// TwinCAT 3 PLC project Library
// Title: lcls-twincat-sample-delivery
// Company: SLAC
// ProjectVersion: 1.0.0
// ProgramVersion: 3.1.4023.0
// libraries:
//   LCLS General, * (SLAC)
//   LCLS Vacuum, * (SLAC - LCLS)
//   PMPS, * (SLAC - LCLS)
//   Tc2_EtherCAT, * (Beckhoff Automation GmbH)
//   Tc2_MC2, * (Beckhoff Automation GmbH)
//   Tc2_ModbusSrv, * (Beckhoff Automation GmbH)
//   Tc2_SerialCom, * (Beckhoff Automation GmbH)
//   Tc2_Standard, * (Beckhoff Automation GmbH)
//   Tc2_SUPS, * (Beckhoff Automation GmbH)
//   Tc2_System, * (Beckhoff Automation GmbH)
//   Tc2_Utilities, * (Beckhoff Automation GmbH)
//   Tc3_Module, * (Beckhoff Automation GmbH)
//   TcUnit, * (www.tcunit.org)
// project tree:
//   DUTs/ALI/ E_AxisMoveMode.TcDUT (not stored), E_CTRL_MODE.TcDUT (not stored), E_PropValveFBState.TcDUT (not stored), HMI_PropValveCtrlState.TcDUT (not stored), ST_ALI.TcDUT (not stored), ST_ManipAxis.TcDUT (not stored), ST_PIDParams.TcDUT (not stored), ST_PressureController.TcDUT (not stored), ST_PropValveMKS253.TcDUT (not stored)
//   DUTs/Bronkhorst/ E_BHElFlowUnit.TcDUT (not stored), ST_BhElFlow.TcDUT (not stored)
//   DUTs/ E_AxisMotionState.TcDUT (not stored), ST_ManifoldValve.TcDUT (not stored), ST_Proportionair.TcDUT (not stored), ST_RegDeadbandControls.TcDUT (not stored), ST_Regulator.TcDUT (not stored), ST_SelectorM3.TcDUT (not stored), ST_Shaker.TcDUT (not stored), ST_ShakerControls.TcDUT (not stored), ST_Strings.TcDUT (not stored)
//   DUTs/General/ E_CTRL_MODE_1.TcDUT
//   DUTs/IO_Structs/ ST_ALIIO.TcDUT (not stored), ST_M3DeviceBaseIO.TcDUT (not stored), ST_SerialComm.TcDUT (not stored)
//   DUTs/Sensirion/ E_SensirionFMMode.TcTLEO (not stored), ST_SensirionFM.TcDUT (not stored), ST_SensirionFMControl.TcDUT (not stored), ST_SensirionFMStatus.TcDUT (not stored)
//   DUTs/TEC/ ST_TECControl.TcDUT (not stored), ST_TECStatus.TcDUT (not stored)
//   DUTs/Vici/ ST_4PViciValveSampleNames.TcDUT, ST_ViciControl.TcDUT (not stored), ST_ViciStatus.TcDUT (not stored)
//   GVLs/ GVL_SAMPLE.TcGVL
//   / PlcTask.TcTTO
//   POUs/ALI/ FB_ALI.TcPOU (not stored), FB_ManipAxis.TcPOU (not stored), FB_PID_EXT.TcPOU (not stored), FB_PropValve.TcPOU (not stored), F_AxisRef_To_MSTA.TcPOU (not stored), MC_SmoothMover.TcPOU (not stored)
//   POUs/Bronkhorst/ FB_BronkhorstMFM.TcPOU (not stored)
//   POUs/DigitalOutput/ FB_SolenoidPair.TcPOU (not stored)
//   POUs/ FB_RCC.TcPOU, EXAMPLE_DEPLOYMENT.TcPOU (not stored), PRG_TEST.TcPOU (not stored)
//   POUs/GasManifold/ FB_GasManifold.TcPOU (not stored), FB_ManiValve.TcPOU (not stored)
//   POUs/Helpers/ FB_EcatDiag.TcPOU (not stored), FB_SelectorSync.TcPOU (not stored), FB_SerialCommWrapper.TcPOU (not stored), FB_ShiftByteArray.TcPOU (not stored)
//   POUs/PCM/ FB_PressureControlModule.TcPOU (not stored)
//   POUs/Regulators/ FB_ProportionairRegulator.TcPOU (not stored), FB_Regulator.TcPOU (not stored), F_rPressure.TcPOU (not stored)
//   POUs/Selectors/ FB_SelectorM3.TcPOU (not stored)
//   POUs/Sensirion/ FB_SensirionDriver.TcPOU, FB_SensirionTransaction.TcPOU (not stored), fSHDLCChecksum.TcPOU (not stored)
//   POUs/TEC/ FB_TECDriver.TcPOU (not stored), FB_TECTransaction.TcPOU (not stored)
//   POUs/Tests/ FB_RCC_TEST.TcPOU
//   POUs/VICI/ FB_4PortViciValve.TcPOU, FB_ViciDriver.TcPOU, FB_ViciTransaction.TcPOU (not stored), FB_ViciValve.TcPOU (not stored)

CONFIGURATION Library
    RESOURCE PLC ON TwinCAT3
        TASK PlcTask(INTERVAL := T#10ms, PRIORITY := 20);
        PROGRAM PRG_TEST WITH PlcTask : PRG_TEST;
    END_RESOURCE
END_CONFIGURATION

// ---- DUTs/General/E_CTRL_MODE_1.TcDUT
{attribute 'qualified_only'}
{attribute 'strict'}
TYPE E_CTRL_MODE_1 :
(
    enum_member := 0
);
END_TYPE

// ---- DUTs/Vici/ST_4PViciValveSampleNames.TcDUT
TYPE ST_4PViciValveSampleNames :
STRUCT
      {attribute 'pytmc' := '
        pv: 01
        io: io
     '}
     s1 : STRING;
     {attribute 'pytmc' := '
        pv: 02
        io: io
     '}
     s2 : STRING;
     {attribute 'pytmc' := '
        pv: 03
        io: io
     '}
     s3 : STRING;
     {attribute 'pytmc' := '
        pv: 04
        io: io
     '}
     s4 : STRING;
END_STRUCT
END_TYPE

// ---- GVLs/GVL_SAMPLE.TcGVL
VAR_GLOBAL
    g_xFirstPass: BOOL := TRUE;
END_VAR

// ---- POUs/FB_RCC.TcPOU
FUNCTION_BLOCK FB_RCC
VAR_IN_OUT
	RCC_VRC_01 : FB_VRC_NC_ClsLS;
	RCC_VRC_02 : FB_VRC;
	RCC_VRC_03 : FB_VRC_NC_ClsLS;
	RCC_VRC_04 : FB_VRC_NC_ClsLS;
	RCC_GCP_01 : FB_901_ECAT;
END_VAR
VAR
	{attribute 'pytmc' :=' pv: ILK_Setpoint '}
    RCC_GCP_01_INTERLOCK_SETPOINT : REAL := 10;
	{attribute 'pytmc' :=' pv: OverrideMode '}
	xSystemOverrideMode_RCC : BOOL := FALSE;
	{attribute 'pytmc' :=' pv: sLogMessage '}
	sLogMessage : T_MaxString := "";
	fbFormat   : FB_FormatString;
	
	tTimer1 : TON;
	current_state : INT := 0;
	start_cycle : BOOL  := FALSE;
	
	RCC_VRC_01_OPEN_OK : BOOL;
    RCC_VRC_02_OPEN_OK : BOOL;
    RCC_VRC_03_OPEN_OK : BOOL;
    RCC_VRC_04_OPEN_OK : BOOL;
END_VAR


(* Valve can open only when CRIX-RCC-VRC-02 and 03 are closed*)
RCC_VRC_01_OPEN_OK := ( RCC_VRC_02.iq_stValve.i_xClsLS AND NOT RCC_VRC_02.iq_stValve.q_xOPN_DO ) AND
                                    ( RCC_VRC_03.iq_stValve.i_xClsLS AND NOT RCC_VRC_03.iq_stValve.q_xOPN_DO ) ;

RCC_VRC_01(i_xExtILK_OK := RCC_VRC_01_OPEN_OK,
                i_xOverrideMode := xSystemOverrideMode_RCC,
                 iq_stValve=> );

(* Valve can open only when CRIX-RCC-VRC-01 and 04 are closed*)
RCC_VRC_02_OPEN_OK := ( RCC_VRC_01.iq_stValve.i_xClsLS AND NOT RCC_VRC_01.iq_stValve.q_xOPN_DO ) AND
                                    ( RCC_VRC_04.iq_stValve.i_xClsLS AND NOT RCC_VRC_04.iq_stValve.q_xOPN_DO );

RCC_VRC_02(i_xExtILK_OK := RCC_VRC_02_OPEN_OK,
                i_xOverrideMode := xSystemOverrideMode_RCC,
                 iq_stValve=> );

(* Valve can open only when CRIX-RCC-GCP-01 reading < setpoint Torr and CRIX-RCC-VRC-01 and 04 are closed*)
RCC_VRC_03_OPEN_OK := (RCC_GCP_01.PG.rPRESS < RCC_GCP_01_INTERLOCK_SETPOINT and RCC_GCP_01.PG.xPRESS_OK ) AND
                                 ( RCC_VRC_01.iq_stValve.i_xClsLS AND NOT RCC_VRC_01.iq_stValve.q_xOPN_DO ) AND
                                              ( RCC_VRC_04.iq_stValve.i_xClsLS AND NOT RCC_VRC_04.iq_stValve.q_xOPN_DO );

RCC_VRC_03(i_xExtILK_OK := RCC_VRC_03_OPEN_OK,
                i_xOverrideMode := xSystemOverrideMode_RCC,
                 iq_stValve=> );

(* Valve can open only when CRIX-RCC-VRC-02 and 03 are closed*)
RCC_VRC_04_OPEN_OK := ( RCC_VRC_02.iq_stValve.i_xClsLS AND NOT RCC_VRC_02.iq_stValve.q_xOPN_DO ) AND
                                      ( RCC_VRC_03.iq_stValve.i_xClsLS AND NOT RCC_VRC_03.iq_stValve.q_xOPN_DO ) ;

RCC_VRC_04(i_xExtILK_OK := RCC_VRC_04_OPEN_OK,
                i_xOverrideMode := xSystemOverrideMode_RCC,
                 iq_stValve=> );

METHOD PUBLIC cycle : BOOL
VAR_INPUT
	t1 : TIME := T#20s;
	t2 : TIME := T#10s;
	t3 : TIME := T#5s;
	t4 : TIME := T#10s;
	run_clean : BOOL := TRUE;
END_VAR
CASE current_state OF
	-1:
		IF start_cycle THEN 
			current_state := 0; 
			start_cycle := FALSE;
		END_IF
		
	0:
		RCC_VRC_01.iq_stValve.q_xOPN_DO := FALSE;
		RCC_VRC_02.iq_stValve.q_xOPN_DO := FALSE;
		RCC_VRC_03.iq_stValve.q_xOPN_DO := FALSE;
		RCC_VRC_04.iq_stValve.q_xOPN_DO := FALSE;
		current_state:=1;
		
	1: // OPEN
		tTimer1(IN:=TRUE, PT:=t1);
		RCC_VRC_02.iq_stValve.q_xOPN_DO := TRUE;
	
		IF tTimer1.Q THEN 
			current_state := 2;
			tTimer1(IN:=FALSE); // RESTART TIMER
		END_IF
		
	2:	// DRAIN_1
		IF RCC_VRC_03_OPEN_OK THEN 
			IF run_clean THEN RCC_VRC_02.iq_stValve.q_xOPN_DO := FALSE; END_IF
			RCC_VRC_03.iq_stValve.q_xOPN_DO := TRUE;
			current_state := 3; 
		END_IF
		
	3:	// DRAIN_2
		tTimer1(IN:=TRUE, PT:=t2);
		
		IF tTimer1.Q THEN 
			current_state := 4;
			IF NOT RCC_VRC_03_OPEN_OK THEN current_state := 1; END_IF
 			RCC_VRC_03.iq_stValve.q_xOPN_DO := FALSE;
			IF NOT run_clean THEN RCC_VRC_02.iq_stValve.q_xOPN_DO := FALSE; END_IF
			tTimer1(IN:=FALSE); // RESTART TIMER
		END_IF
		
	4: // OPEN VRC_01 for T3
		tTimer1(IN:=TRUE, PT:=t3);
		RCC_VRC_01.iq_stValve.q_xOPN_DO := TRUE;
		IF tTimer1.Q THEN 
			current_state := 5;
			tTimer1(IN:=FALSE); // RESTART TIMER
		END_IF
		
	5: // OPEN VRC_04 for T4
		tTimer1(IN:=TRUE, PT:=t4);
		RCC_VRC_04.iq_stValve.q_xOPN_DO := TRUE;
		IF tTimer1.Q THEN 
			current_state := -1;
			RCC_VRC_01.iq_stValve.q_xOPN_DO := FALSE;
			RCC_VRC_04.iq_stValve.q_xOPN_DO := FALSE;
			tTimer1(IN:=FALSE); // RESTART TIMER
		END_IF	
	
	
END_CASE
END_METHOD

END_FUNCTION_BLOCK

// ---- POUs/Sensirion/FB_SensirionDriver.TcPOU
FUNCTION_BLOCK FB_SensirionDriver

VAR_INPUT
    i_xExecute				: BOOL := FALSE;		(* rising edge execute *)
    i_tTimeOut				: TIME := T#10S;  		(* Maximum wait time for reply *)
    i_stControl				: ST_SensirionFMControl;
END_VAR
VAR_OUTPUT
    q_xDone					: BOOL;
    q_xError				: BOOL;
    q_xWarning				: BOOL;					(* set in the event of an unexpected reply *)
    q_xTimeout				: BOOL;
    q_asResult				: ARRAY[1..60] OF STRING(255);
    q_stStatus				: ST_SensirionFMStatus;
    q_xInitComplete			: BOOL;
END_VAR
VAR_IN_OUT
    iq_stSerialRXBuffer 	: ComBuffer;
    iq_stSerialTXBuffer 	: ComBuffer;
END_VAR
VAR
    //Usual stuff
    rtExecute				: R_TRIG;
    rtReInit				:	R_TRIG;
    iStep					: INT;
    iResultIndex			:	INT := 1;
    aiSteps	:	ARRAY[1..256] OF INT;
    iStepIndex	:	INT;
    fbSensirionTransaction		: FB_SensirionTransaction;

    //Device Specific Working Variables
    tonDelay : TON;
    bLen	:	BYTE;
    abTxData	:	ARRAY[1..256] OF BYTE;
    xInitComplete	:	BOOL;
    abRxData	:	ARRAY[1..256] OF BYTE;

    iScale	:	INT;
    iUnit	:	INT;
    xType	:	BOOL;
    xMode	:	BYTE;
    xLinear	:	BOOL;
    uiOffset	:	UINT;
    iIdleAttempt : INT;

    //Command delays
    tonCommandDelay : TON;
xcatch : BOOL;
END_VAR

(* This function block performs serial communication with a Sensirion meter *)


(* rising edge trigger *)
rtExecute(CLK:= i_xExecute);
rtReInit(CLK:= i_stControl.xReset);
IF rtReInit.Q THEN xInitComplete := FALSE; END_IF
IF rtExecute.Q  THEN
    q_xDone	:= FALSE;
    q_xError := FALSE;
    q_xWarning := FALSE;
    q_xTimeout := FALSE;
    q_asResult[iResultIndex]:= '';
    fbSensirionTransaction( i_xExecute:= FALSE, iq_stSerialRXBuffer:= iq_stSerialRXBuffer, iq_stSerialTXBuffer:= iq_stSerialTXBuffer );  (* reset *)
    IF xInitComplete THEN
        iStep := 30;
        (* Branch to reset device if reset bit is set here *)
        IF rtReInit.Q  OR (i_stControl.xCalMode <> q_stStatus.xFMMode) THEN
            iStep := 400;
            xInitComplete := FALSE;
            q_stStatus.xFlowValid := FALSE;
            q_asResult[iResultIndex] := 'Reinitializing';
            iResultIndex := iResultIndex +1;
        END_IF
    ELSIF i_stControl.xReset THEN
        iStep := 400;
        q_stStatus.xFlowValid := FALSE;
        q_asResult[iResultIndex] := 'Reinitializing';
        iResultIndex := iResultIndex +1;
    ELSE
        iStep := 9;
    END_IF
END_IF

CASE iStep OF
    0: (* idle *)
        ;

    9: //Get cal mode
    fbSensirionTransaction(
        i_xExecute:= TRUE,
        i_bAdr:= i_stControl.bAdr,
        i_bLen:= 0,
        i_bCmd:= 16#43,
        i_abTxData := abTxData,
        i_tTimeOut:= i_tTimeOut,
        iq_stSerialRXBuffer:= iq_stSerialRXBuffer,
        iq_stSerialTXBuffer:= iq_stSerialTXBuffer
        );
    IF fbSensirionTransaction.q_xError THEN
        q_asResult[iResultIndex] := CONCAT('in Step 9 serial transaction failed with message: ', fbSensirionTransaction.q_sResult);
        iResultIndex := iResultIndex +1;
        iStep := 9000;
    ELSIF fbSensirionTransaction.q_xDone THEN
        //abRxdata := fbSensirionTransaction.q_baRxData;
        IF UDINT_TO_BOOL(MEMCPY(destAddr:=ADR(xMode), srcAddr:=ADR(fbSensirionTransaction.q_baRxData), n:=1)) THEN
            q_stStatus.xFMMode := BYTE_TO_BOOL(xMode);
            fbSensirionTransaction( i_xExecute:= FALSE, iq_stSerialRXBuffer:= iq_stSerialRXBuffer, iq_stSerialTXBuffer:= iq_stSerialTXBuffer );  (* reset *)
            q_asResult[iResultIndex] := CONCAT('Step 9 complete. Cal mode is set to: ', BYTE_TO_STRING(xMode));
            iResultIndex := iResultIndex +1;
        ELSE
            iStep := 9000;
            q_asResult[iResultIndex] := 'Memcpy in step 9 failed';
            iResultIndex := iResultIndex +1;
        END_IF
        iStep := 10;
    END_IF

    10: // Set calibration
    //calibration of 0 for precision mode, 250 nL/min - 5000 nL/min
    // calibration of 1 for extended mode, 2000 nL/min - 20000 nL/min
    IF q_stStatus.xFMMode <> i_stControl.xCalMode THEN
        IF i_stControl.xCalMode THEN abTxData[1]:=1; ELSE abTxData[1]:=0; END_IF
        fbSensirionTransaction(
            i_xExecute:= TRUE,
            i_bAdr:= i_stControl.bAdr,
            i_bLen:= 1,
            i_bCmd:= 16#43,
            i_abTxData := abTxData,
            i_tTimeOut:= i_tTimeOut,
            iq_stSerialRXBuffer:= iq_stSerialRXBuffer,
            iq_stSerialTXBuffer:= iq_stSerialTXBuffer
            );
        IF fbSensirionTransaction.q_xError THEN
            q_asResult[iResultIndex] := CONCAT('in Step 10 serial transaction failed with message: ', fbSensirionTransaction.q_sResult);
            iResultIndex := iResultIndex +1;
            iStep := 9000;
        ELSIF fbSensirionTransaction.q_xDone THEN
            tonCommandDelay(IN:=fbSensirionTransaction.q_xDone, PT:=T#1S);
            IF tonCommandDelay.Q THEN
                (* No response, completed transaction confirmed by a response*)
                q_asResult[iResultIndex] := 'Step 10 complete';
                iResultIndex := iResultIndex +1;
                iStep := 11;
                fbSensirionTransaction( i_xExecute:= FALSE, iq_stSerialRXBuffer:= iq_stSerialRXBuffer, iq_stSerialTXBuffer:= iq_stSerialTXBuffer );  (* reset *)
            END_IF
        END_IF
    ELSE
        q_asResult[iResultIndex] := 'Calmode already set';
        iResultIndex := iResultIndex +1;
        iStep := 11;
    END_IF

    11: //Get cal mode
    fbSensirionTransaction(
        i_xExecute:= TRUE,
        i_bAdr:= i_stControl.bAdr,
        i_bLen:= 0,
        i_bCmd:= 16#43,
        i_abTxData := abTxData,
        i_tTimeOut:= i_tTimeOut,
        iq_stSerialRXBuffer:= iq_stSerialRXBuffer,
        iq_stSerialTXBuffer:= iq_stSerialTXBuffer
        );
    IF fbSensirionTransaction.q_xError THEN
        q_asResult[iResultIndex] := CONCAT('in Step 11 serial transaction failed with message: ', fbSensirionTransaction.q_sResult);
        iResultIndex := iResultIndex +1;
        iStep := 9000;
    ELSIF fbSensirionTransaction.q_bState <> 0 THEN
        q_asResult[iResultIndex] := CONCAT('in Step 11 serial transaction failed with error state: ', BYTE_TO_STRING(fbSensirionTransaction.q_bState));
        iResultIndex := iResultIndex +1;
        fbSensirionTransaction( i_xExecute:= FALSE, iq_stSerialRXBuffer:= iq_stSerialRXBuffer, iq_stSerialTXBuffer:= iq_stSerialTXBuffer );  (* reset *)
        iStep := 9000;
    ELSIF fbSensirionTransaction.q_xDone THEN
        tonCommandDelay(IN:=fbSensirionTransaction.q_xDone, PT:=T#100MS);
        IF tonCommandDelay.Q THEN
            IF UDINT_TO_BOOL(MEMCPY(destAddr:=ADR(xMode), srcAddr:=ADR(fbSensirionTransaction.q_baRxData), n:=1)) THEN
                q_stStatus.xFMMode := BYTE_TO_BOOL(xMode);
                fbSensirionTransaction( i_xExecute:= FALSE, iq_stSerialRXBuffer:= iq_stSerialRXBuffer, iq_stSerialTXBuffer:= iq_stSerialTXBuffer );  (* reset *)
                q_asResult[iResultIndex] := 'Step 11 complete';
                iResultIndex := iResultIndex +1;
                iStep := 12;
            ELSE
                iStep := 9000;
                q_asResult[iResultIndex] := 'Memcpy in step 9 failed';
                iResultIndex := iResultIndex +1;
            END_IF
        END_IF
    END_IF

    12: //Get scale factor
    fbSensirionTransaction(
        i_xExecute:= TRUE,
        i_bAdr:= i_stControl.bAdr,
        i_bLen:= 0,
        i_bCmd:= 16#53,
        i_abTxData := abTxData,
        i_tTimeOut:= i_tTimeOut,
        iq_stSerialRXBuffer:= iq_stSerialRXBuffer,
        iq_stSerialTXBuffer:= iq_stSerialTXBuffer
        );
    IF fbSensirionTransaction.q_xError THEN
        q_asResult[iResultIndex] := CONCAT('in Step 12 serial transaction failed with message: ', fbSensirionTransaction.q_sResult);
        iResultIndex := iResultIndex +1;
        iStep := 9000;
    ELSIF fbSensirionTransaction.q_bState <> 0 THEN
        q_asResult[iResultIndex] := CONCAT('in Step 12 serial transaction failed with error state: ', BYTE_TO_STRING(fbSensirionTransaction.q_bState));
        iResultIndex := iResultIndex +1;
        fbSensirionTransaction( i_xExecute:= FALSE, iq_stSerialRXBuffer:= iq_stSerialRXBuffer, iq_stSerialTXBuffer:= iq_stSerialTXBuffer );  (* reset *)
        iStep := 9000;
    ELSIF fbSensirionTransaction.q_xDone THEN
        tonCommandDelay(IN:=fbSensirionTransaction.q_xDone, PT:=T#100MS);
        IF tonCommandDelay.Q THEN
            IF UDINT_TO_BOOL(MEMCPY(destAddr:=ADR(iScale), srcAddr:=ADR(fbSensirionTransaction.q_baRxData), n:=2)) THEN //always 2 for the 16 bit wide integer
                iScale := WORD_TO_INT(HOST_TO_BE16(INT_TO_WORD(iScale)));
                fbSensirionTransaction( i_xExecute:= FALSE, iq_stSerialRXBuffer:= iq_stSerialRXBuffer, iq_stSerialTXBuffer:= iq_stSerialTXBuffer );  (* reset *)
                q_asResult[iResultIndex] := 'Step 12 complete';
                iResultIndex := iResultIndex +1;
                iStep := 13;
            ELSE
                iStep := 9000;
                q_asResult[iResultIndex] := 'Memcpy in step 12 failed';
                iResultIndex := iResultIndex +1;
            END_IF
        END_IF
    END_IF

    13: //Get flow unit
    fbSensirionTransaction(
        i_xExecute:= TRUE,
        i_bAdr:= i_stControl.bAdr,
        i_bLen:= 0,
        i_bCmd:= 16#52,
        i_abTxData := abTxData,
        i_tTimeOut:= i_tTimeOut,
        iq_stSerialRXBuffer:= iq_stSerialRXBuffer,
        iq_stSerialTXBuffer:= iq_stSerialTXBuffer
        );
    IF fbSensirionTransaction.q_xError THEN
        q_asResult[iResultIndex] := CONCAT('in Step 13 serial transaction failed with message: ', fbSensirionTransaction.q_sResult);
        iResultIndex := iResultIndex +1;
        iStep := 9000;
    ELSIF fbSensirionTransaction.q_bState <> 0 THEN
        q_asResult[iResultIndex] := CONCAT('in Step 13 serial transaction failed with error state: ', BYTE_TO_STRING(fbSensirionTransaction.q_bState));
        iResultIndex := iResultIndex +1;
        fbSensirionTransaction( i_xExecute:= FALSE, iq_stSerialRXBuffer:= iq_stSerialRXBuffer, iq_stSerialTXBuffer:= iq_stSerialTXBuffer );  (* reset *)
        iStep := 9000;
    ELSIF fbSensirionTransaction.q_xDone THEN
        tonCommandDelay(IN:=fbSensirionTransaction.q_xDone, PT:=T#100MS);
        IF tonCommandDelay.Q THEN
            IF UDINT_TO_BOOL(MEMCPY(destAddr:=ADR(iUnit), srcAddr:=ADR(fbSensirionTransaction.q_baRxData), n:=2)) THEN //always 2 for the 16 bit wide integer
                iUnit := WORD_TO_INT(HOST_TO_BE16(INT_TO_WORD(iUnit)));
                fbSensirionTransaction( i_xExecute:= FALSE, iq_stSerialRXBuffer:= iq_stSerialRXBuffer, iq_stSerialTXBuffer:= iq_stSerialTXBuffer );  (* reset *)
                q_asResult[iResultIndex] := 'Step 13 complete';
                iResultIndex := iResultIndex +1;
                iStep := 14;
            ELSE
                iStep := 9000;
                q_asResult[iResultIndex] := 'Memcpy in step 13 failed';
                iResultIndex := iResultIndex +1;
            END_IF
        END_IF
    END_IF

    14: //Get measurement type
    fbSensirionTransaction(
        i_xExecute:= TRUE,
        i_bAdr:= i_stControl.bAdr,
        i_bLen:= 0,
        i_bCmd:= 16#55,
        i_abTxData := abTxData,
        i_tTimeOut:= i_tTimeOut,
        iq_stSerialRXBuffer:= iq_stSerialRXBuffer,
        iq_stSerialTXBuffer:= iq_stSerialTXBuffer
        );
    IF fbSensirionTransaction.q_xError THEN
        q_asResult[iResultIndex] := CONCAT('in Step 14 serial transaction failed with message: ', fbSensirionTransaction.q_sResult);
        iResultIndex := iResultIndex +1;
        iStep := 9000;
    ELSIF fbSensirionTransaction.q_bState <> 0 THEN
        q_asResult[iResultIndex] := CONCAT('in Step 14 serial transaction failed with error state: ', BYTE_TO_STRING(fbSensirionTransaction.q_bState));
        iResultIndex := iResultIndex +1;
        fbSensirionTransaction( i_xExecute:= FALSE, iq_stSerialRXBuffer:= iq_stSerialRXBuffer, iq_stSerialTXBuffer:= iq_stSerialTXBuffer );  (* reset *)
        iStep := 9000;
    ELSIF fbSensirionTransaction.q_xDone THEN
        tonCommandDelay(IN:=fbSensirionTransaction.q_xDone, PT:=T#100MS);
        IF tonCommandDelay.Q THEN
            xType := BYTE_TO_BOOL(fbSensirionTransaction.q_baRxData[1]);
            q_asResult[iResultIndex] := 'Step 14 complete';
            iResultIndex := iResultIndex +1;
            iStep := 16;
            fbSensirionTransaction( i_xExecute:= FALSE, iq_stSerialRXBuffer:= iq_stSerialRXBuffer, iq_stSerialTXBuffer:= iq_stSerialTXBuffer );  (* reset *)
        END_IF
    END_IF

    15: //Get offset
    fbSensirionTransaction(
        i_xExecute:= TRUE,
        i_bAdr:= i_stControl.bAdr,
        i_bLen:= 0,
        i_bCmd:= 16#56,
        i_abTxData := abTxData,
        i_tTimeOut:= i_tTimeOut,
        iq_stSerialRXBuffer:= iq_stSerialRXBuffer,
        iq_stSerialTXBuffer:= iq_stSerialTXBuffer
        );
    IF fbSensirionTransaction.q_xError THEN
        q_asResult[iResultIndex] := CONCAT('in Step 15 serial transaction failed with message: ', fbSensirionTransaction.q_sResult);
        iResultIndex := iResultIndex +1;
        iStep := 9000;
    ELSIF fbSensirionTransaction.q_bState <> 0 THEN
        q_asResult[iResultIndex] := CONCAT('in Step 15 serial transaction failed with error state: ', BYTE_TO_STRING(fbSensirionTransaction.q_bState));
        iResultIndex := iResultIndex +1;
        fbSensirionTransaction( i_xExecute:= FALSE, iq_stSerialRXBuffer:= iq_stSerialRXBuffer, iq_stSerialTXBuffer:= iq_stSerialTXBuffer );  (* reset *)
        iStep := 9000;
    ELSIF fbSensirionTransaction.q_xDone THEN
        tonCommandDelay(IN:=fbSensirionTransaction.q_xDone, PT:=T#100MS);
        IF tonCommandDelay.Q THEN
            IF UDINT_TO_BOOL(MEMCPY(destAddr:=ADR(uiOffset), srcAddr:=ADR(fbSensirionTransaction.q_baRxData), n:=2)) THEN //always 2 for the 16 bit wide integer
                uiOffset := WORD_TO_UINT(HOST_TO_BE16(UINT_TO_WORD(uiOffset)));
                A_ClearTransaction();  (* reset *)
                q_asResult[iResultIndex] := CONCAT('Step 15 complete, offset is: ', UINT_TO_STRING(uiOffset));
                iResultIndex := iResultIndex +1;
                iStep := 16;
            ELSE
                iStep := 9000;
                q_asResult[iResultIndex] := 'Memcpy in step 15 failed';
                iResultIndex := iResultIndex +1;
            END_IF
            A_ClearTransaction();  (* reset *)
        END_IF
    END_IF

    16: //Get linear mode
    fbSensirionTransaction(
        i_xExecute:= TRUE,
        i_bAdr:= i_stControl.bAdr,
        i_bLen:= 0,
        i_bCmd:= 16#45,
        i_abTxData := abTxData,
        i_tTimeOut:= i_tTimeOut,
        iq_stSerialRXBuffer:= iq_stSerialRXBuffer,
        iq_stSerialTXBuffer:= iq_stSerialTXBuffer
        );
    IF fbSensirionTransaction.q_xError THEN
        q_asResult[iResultIndex] := CONCAT('in Step 16 serial transaction failed with message: ', fbSensirionTransaction.q_sResult);
        iResultIndex := iResultIndex +1;
        iStep := 9000;
    ELSIF fbSensirionTransaction.q_bState <> 0 THEN
        q_asResult[iResultIndex] := CONCAT('in Step 16 serial transaction failed with error state: ', BYTE_TO_STRING(fbSensirionTransaction.q_bState));
        iResultIndex := iResultIndex +1;
        fbSensirionTransaction( i_xExecute:= FALSE, iq_stSerialRXBuffer:= iq_stSerialRXBuffer, iq_stSerialTXBuffer:= iq_stSerialTXBuffer );  (* reset *)
        iStep := 9000;
    ELSIF fbSensirionTransaction.q_xDone THEN
        tonCommandDelay(IN:=fbSensirionTransaction.q_xDone, PT:=T#100MS);
        IF tonCommandDelay.Q THEN
            xLinear := BYTE_TO_BOOL(fbSensirionTransaction.q_baRxData[1]);
            A_ClearTransaction();  (* reset *)
            q_asResult[iResultIndex] := CONCAT('Step 16 complete, linear is: ', BOOL_TO_STRING(xLinear));
            iResultIndex := iResultIndex +1;
            iStep := 20;
        END_IF
    END_IF

//////////////////////////////////////////////////////////////////
// Reset sequence
//////////////////////////////////////////////////////////////////
(*
1. Issue a stop command to halt continuous measurement
2. Reset command
3. Reset initcomplete bit, and xReset
4. Move to done state
*)

    400: //Stop measurement
    fbSensirionTransaction(
        i_xExecute:= TRUE,
        i_bAdr:= i_stControl.bAdr,
        i_bLen:= 0,
        i_bCmd:= 16#34,
        i_abTxData := abTxData,
        i_tTimeOut:= i_tTimeOut,
        iq_stSerialRXBuffer:= iq_stSerialRXBuffer,
        iq_stSerialTXBuffer:= iq_stSerialTXBuffer
        );
    IF fbSensirionTransaction.q_xError THEN
        q_asResult[iResultIndex] := CONCAT('in Step 400 serial transaction failed with message: ', fbSensirionTransaction.q_sResult);
        iResultIndex := iResultIndex +1;
        iStep := 9000;
    ELSIF fbSensirionTransaction.q_xDone THEN
        tonCommandDelay(IN:=fbSensirionTransaction.q_xDone, PT:=T#250MS);
        IF tonCommandDelay.Q THEN
            q_asResult[iResultIndex] := 'Measurement stop command sent';
            iResultIndex := iResultIndex +1;
            iStep:=405;
            fbSensirionTransaction( i_xExecute:= FALSE, iq_stSerialRXBuffer:= iq_stSerialRXBuffer, iq_stSerialTXBuffer:= iq_stSerialTXBuffer );  (* reset *)
        END_IF
    END_IF

    405: //Check sensor status
    fbSensirionTransaction(
        i_xExecute:= TRUE,
        i_bAdr:= i_stControl.bAdr,
        i_bLen:= 0,
        i_bCmd:= 16#30,
        i_abTxData := abTxData,
        i_tTimeOut:= i_tTimeOut,
        iq_stSerialRXBuffer:= iq_stSerialRXBuffer,
        iq_stSerialTXBuffer:= iq_stSerialTXBuffer
        );
    IF fbSensirionTransaction.q_xError THEN
        q_asResult[iResultIndex] := CONCAT('in Step 405 serial transaction failed with message: ', fbSensirionTransaction.q_sResult);
        iResultIndex := iResultIndex +1;
        iStep := 9000;
    ELSIF fbSensirionTransaction.q_xDone THEN
        (* The status measurement is available at the rx data here *)
        IF fbSensirionTransaction.q_iRxLen > 0 THEN
            IF UDINT_TO_BOOL(MEMCPY(destAddr:=ADR(q_stStatus.bStatus), srcAddr:=ADR(fbSensirionTransaction.q_baRxData), n:=1)) THEN
                IF q_stStatus.bStatus.0 = 0 THEN //lsb of bStatus is idle
                    iStep :=410;
                    q_asResult[iResultIndex] := 'Sensor is idle.';
                    iResultIndex := iResultIndex +1;
                    fbSensirionTransaction( i_xExecute:= FALSE, iq_stSerialRXBuffer:= iq_stSerialRXBuffer, iq_stSerialTXBuffer:= iq_stSerialTXBuffer );  (* reset *)
                ELSE
                    iStep := 400;
                    iIdleAttempt := iIdleAttempt + 1;
                    q_asResult[iResultIndex +1] := CONCAT('Failed to move to idle state in step 405, attempt ' , CONCAT(INT_TO_STRING(iIdleAttempt) , ' of 3'));
                    IF iIdleAttempt = 3 THEN iStep := 9000; iIdleAttempt := 0; END_IF
                    fbSensirionTransaction( i_xExecute:= FALSE, iq_stSerialRXBuffer:= iq_stSerialRXBuffer, iq_stSerialTXBuffer:= iq_stSerialTXBuffer );  (* reset *)
                END_IF
            ELSE
                iStep := 9000;
                q_asResult[iResultIndex] := 'Memcpy in step 405 failed';
                iResultIndex := iResultIndex +1;
            END_IF
        ELSE
            q_asResult[iResultIndex] := 'No status data returned';
            iResultIndex := iResultIndex +1;
            iStep := 9000;
        END_IF
    END_IF

    410: //Reset device
    fbSensirionTransaction(
        i_xExecute:= TRUE,
        i_bAdr:= i_stControl.bAdr,
        i_bLen:= 0,
        i_bCmd:= 16#65,
        i_abTxData := abTxData,
        i_tTimeOut:= i_tTimeOut,
        iq_stSerialRXBuffer:= iq_stSerialRXBuffer,
        iq_stSerialTXBuffer:= iq_stSerialTXBuffer
        );
    IF fbSensirionTransaction.q_xError THEN
        q_asResult[iResultIndex] := CONCAT('in Step 400 serial transaction failed with message: ', fbSensirionTransaction.q_sResult);
        iResultIndex := iResultIndex +1;
        iStep := 9000;
    ELSIF fbSensirionTransaction.q_xDone THEN
        tonCommandDelay(IN:=fbSensirionTransaction.q_xDone, PT:=T#200MS);
        IF tonCommandDelay.Q THEN
            q_asResult[iResultIndex] := 'Device reset command sent';
            iResultIndex := iResultIndex +1;
            iStep:=8000;
            xInitComplete := FALSE;
            fbSensirionTransaction( i_xExecute:= FALSE, iq_stSerialRXBuffer:= iq_stSerialRXBuffer, iq_stSerialTXBuffer:= iq_stSerialTXBuffer );  (* reset *)
        END_IF
    END_IF


    20: //Start continuous measurement
    abTxData[1]:=0;
    abTxData[2]:=0;
        fbSensirionTransaction(
            i_xExecute:= TRUE,
            i_bAdr:= i_stControl.bAdr,
            i_bLen:= 2,
            i_bCmd:= 16#33,
            i_abTxData := abTxData,
            i_tTimeOut:= i_tTimeOut,
            iq_stSerialRXBuffer:= iq_stSerialRXBuffer,
            iq_stSerialTXBuffer:= iq_stSerialTXBuffer
            );
        IF fbSensirionTransaction.q_xError THEN
            q_asResult[iResultIndex] := CONCAT('in Step 20 serial transaction failed with message: ', fbSensirionTransaction.q_sResult);
            iResultIndex := iResultIndex +1;
            iStep := 9000;
        ELSIF fbSensirionTransaction.q_xDone THEN
            tonCommandDelay(IN:=fbSensirionTransaction.q_xDone, PT:=T#250MS);
            IF tonCommandDelay.Q THEN
                (* No response, completed transaction confirmed by a response*)
                iStep := 21;
                q_asResult[iResultIndex] := CONCAT('Sent start measurement command', fbSensirionTransaction.q_sResult);
                iResultIndex := iResultIndex +1;
                fbSensirionTransaction( i_xExecute:= FALSE, iq_stSerialRXBuffer:= iq_stSerialRXBuffer, iq_stSerialTXBuffer:= iq_stSerialTXBuffer );  (* reset *)
            END_IF
        END_IF

    21: //Check sensor status
    fbSensirionTransaction(
        i_xExecute:= TRUE,
        i_bAdr:= i_stControl.bAdr,
        i_bLen:= 0,
        i_bCmd:= 16#30,
        i_abTxData := abTxData,
        i_tTimeOut:= i_tTimeOut,
        iq_stSerialRXBuffer:= iq_stSerialRXBuffer,
        iq_stSerialTXBuffer:= iq_stSerialTXBuffer
        );
    IF fbSensirionTransaction.q_xError THEN
        q_asResult[iResultIndex] := CONCAT('in Step 21 serial transaction failed with message: ', fbSensirionTransaction.q_sResult);
        iResultIndex := iResultIndex +1;
        iStep := 9000;
    ELSIF fbSensirionTransaction.q_xDone THEN
        (* The status measurement is available at the rx data here *)
        IF fbSensirionTransaction.q_iRxLen > 0 THEN
            IF UDINT_TO_BOOL(MEMCPY(destAddr:=ADR(q_stStatus.bStatus), srcAddr:=ADR(fbSensirionTransaction.q_baRxData), n:=1)) THEN
                IF q_stStatus.bStatus.1 = 1 THEN
                    iStep :=30;
                    xInitComplete	:= TRUE;
                    q_asResult[iResultIndex] := 'Init success, sensor is measuring.';
                    iResultIndex := iResultIndex +1;
                    fbSensirionTransaction( i_xExecute:= FALSE, iq_stSerialRXBuffer:= iq_stSerialRXBuffer, iq_stSerialTXBuffer:= iq_stSerialTXBuffer );  (* reset *)
                ELSIF q_stStatus.bStatus.0 = 1 THEN
                    iStep :=21; // if the sensor is busy, and not yet measuring, perhaps we try again
                    q_asResult[iResultIndex] := 'Sensor is busy...';
                    iResultIndex := iResultIndex +1;
                    fbSensirionTransaction( i_xExecute:= FALSE, iq_stSerialRXBuffer:= iq_stSerialRXBuffer, iq_stSerialTXBuffer:= iq_stSerialTXBuffer );  (* reset *)
                ELSE
                    iStep := 9000;
                    q_asResult[iResultIndex +1] := 'Failed to start cont. measurement in step 21';
                END_IF
            ELSE
                iStep := 9000;
                q_asResult[iResultIndex] := 'Memcpy in step 21 failed';
                iResultIndex := iResultIndex +1;
            END_IF
        ELSE
            q_asResult[iResultIndex] := 'No status data returned in step 21';
            iResultIndex := iResultIndex +1;
            iStep := 9000;
        END_IF
    END_IF

    30: //Get last measurement
        tonDelay.IN:=TRUE;
        abTxData[1]:=0;
        fbSensirionTransaction(
        i_xExecute:= tonDelay.Q,
        i_bAdr:= i_stControl.bAdr,
        i_bLen:= 1,
        i_bCmd:= 16#35,
        i_abTxData := abTxData,
        i_tTimeOut:= i_tTimeOut,
        iq_stSerialRXBuffer:= iq_stSerialRXBuffer,
        iq_stSerialTXBuffer:= iq_stSerialTXBuffer
        );
    IF fbSensirionTransaction.q_xError THEN
        q_asResult[iResultIndex] := CONCAT('in Step 30 serial transaction failed with message: ', fbSensirionTransaction.q_sResult);
        iResultIndex := iResultIndex +1;
        iStep := 9000;
    ELSIF fbSensirionTransaction.q_xDone THEN
        (* The flow measurement is available at the rx data here *)
        IF fbSensirionTransaction.q_iRxLen > 0 THEN
            IF UDINT_TO_BOOL(MEMCPY(destAddr:=ADR(q_stStatus.uiSensorOutput), srcAddr:=ADR(fbSensirionTransaction.q_baRxData), n:=2)) THEN //always 2 for the 16 bit wide integer
                q_stStatus.uiSensorOutput := WORD_TO_UINT(HOST_TO_BE16(UINT_TO_WORD(q_stStatus.uiSensorOutput))); //memcpy effs up an produces a little endian number, sensirion transmits be
                IF (q_stStatus.uiSensorOutput AND 32768) = 32768 THEN
                    q_stStatus.iFlowTicks := UINT_TO_INT(-1*((q_stStatus.uiSensorOutput XOR 65535) + 1));
                ELSE
                    q_stStatus.iFlowTicks := UINT_TO_INT(q_stStatus.uiSensorOutput);
                END_IF
                //Conversion from int to real value using the unit
                IF ((INT_TO_WORD(iUnit) AND 16#000F)=16#0003) OR ((INT_TO_WORD(iUnit) AND 16#000F)=16#0004) THEN //lsb of iUnit is magnitude, should only be one thing

                    q_stStatus.rFlow := (INT_TO_REAL(q_stStatus.iFlowTicks)/INT_TO_REAL(iScale))*EXPT(10,-3); //converting from nL to uL

                    (* Check flow readback against calibration range for OoR *)
                    //calibration of 0 for precision mode, 250 nL/min - 5000 nL/min
                    // calibration of 1 for extended mode, 2000 nL/min - 20000 nL/min
                    IF (q_stStatus.xFMMode =0 ) THEN
                        IF (ABS(q_stStatus.rFlow) < (250E-3)) THEN
                            q_stStatus.iState := 2; //<OoR
                        ELSIF (ABS(q_stStatus.rFlow) > (5000E-3)) THEN
                            q_stStatus.iState := 1; //OoR>
                        ELSE
                            q_stStatus.iState := 0; //OK
                        END_IF
                    ELSIF (q_stStatus.xFMMode =1 ) THEN
                        IF (ABS(q_stStatus.rFlow) < (2000E-3)) THEN
                            q_stStatus.iState := 2; //<OoR Add to xOoR variable
                        ELSIF (ABS(q_stStatus.rFlow) > (20000E-3)) THEN
                            q_stStatus.iState := 1; //OoR>
                        ELSE
                            q_stStatus.iState := 0; // OK
                        END_IF
                    END_IF
                    q_stStatus.xFlowValid := (q_stStatus.iState = 0); // Flow valid if OK

                    // Limit the measured flowrate based on the calmode
                    IF q_stStatus.xFMMode THEN
                        q_stStatus.rFlow := LIMIT(-20000E-3, q_stStatus.rFlow, 20000E-3);
                    ELSE
                        q_stStatus.rFlow := LIMIT(-5000E-3, q_stStatus.rFlow, 5000E-3);
                    END_IF

                ELSE
                    iStep := 9000;
                    q_asResult[iResultIndex] := 'iUnit not recognized in step 30';
                    iResultIndex := iResultIndex +1;
                END_IF
                (* Stuff worked, go to 8000 *)
                iStep := 8000;
                fbSensirionTransaction( i_xExecute:= FALSE, iq_stSerialRXBuffer:= iq_stSerialRXBuffer, iq_stSerialTXBuffer:= iq_stSerialTXBuffer );  (* reset *)
                tonDelay.IN := FALSE;
            ELSE
                iStep := 9000;
                q_asResult[iResultIndex] := 'Memcpy in step 30 failed';
                iResultIndex := iResultIndex +1;
            END_IF
        ELSE
            q_asResult[iResultIndex] := 'No flow data returned';
            iResultIndex := iResultIndex +1;
            iStep := 9000;
        END_IF
    END_IF

    8000: (* done *)
        q_xDone := TRUE;
        IF q_asResult[iResultIndex] = '' THEN
            q_asResult[iResultIndex] := 'Success';
            iResultIndex := iResultIndex +1;

        END_IF
        IF  i_xExecute = FALSE THEN
            q_xDone:= FALSE;
            iStep := 0;
        END_IF

    9000:
        q_xTimeout := fbSensirionTransaction.q_xTimeout;
        q_xError := TRUE;
        // If we're having issues communicating we don't want to be left thinking there's a flow... even if we know it's not valid.
        q_stStatus.xFlowValid := FALSE;
        q_stStatus.iState := 3; // Flow invalid
        q_stStatus.rFlow := 0;
END_CASE

tonDelay(PT:=T#500MS);

//q_stStatus.rFlow := INT_TO_REAL(iFlow);
iStepIndex := iStepIndex +1;
aiSteps[iStepIndex]:=iStep;


q_xInitComplete := xInitComplete;

IF iStepIndex >256 THEN iStepIndex:=1; END_IF
IF iResultIndex >60 THEN iResultIndex:=1; END_IF

ACTION A_ClearTransaction:
fbSensirionTransaction( i_xExecute:= FALSE, iq_stSerialRXBuffer:= iq_stSerialRXBuffer, iq_stSerialTXBuffer:= iq_stSerialTXBuffer );  (* reset *)
END_ACTION

ACTION Get:

END_ACTION

METHOD Reset
VAR_INPUT
END_VAR
// If this works....

THIS^(i_xExecute := False,
    iq_stSerialRXBuffer := THIS^.iq_stSerialRXBuffer,
    iq_stSerialTXBuffer := THIS^.iq_stSerialTXBuffer,);
END_METHOD

END_FUNCTION_BLOCK

// ---- POUs/Tests/FB_RCC_TEST.TcPOU
FUNCTION_BLOCK FB_RCC_TEST EXTENDS FB_TestSuite
VAR_INPUT
END_VAR
VAR_OUTPUT
END_VAR
VAR
END_VAR

END_FUNCTION_BLOCK

// ---- POUs/VICI/FB_4PortViciValve.TcPOU
FUNCTION_BLOCK FB_4PortViciValve
VAR_INPUT
    iAdress : INT;
END_VAR
VAR_OUTPUT
END_VAR
VAR
    fbNporValve : FB_ViciValve;
    iNumPorts : INT := 4;

    {attribute 'pytmc' := '
        pv: iReqPos
        io: io
     '}
    iReqPos : INT;
    {attribute 'pytmc' := '
        pv: SampleNames
        io: io
     '}
    stSampleNames : ST_4PViciValveSampleNames;
END_VAR

fbNporValve(iAddress := iAdress, iNumOfPorts := iNumPorts, iReqPos := iReqPos);

END_FUNCTION_BLOCK

// ---- POUs/VICI/FB_ViciDriver.TcPOU
FUNCTION_BLOCK FB_ViciDriver
VAR_INPUT
    i_xExecute				: BOOL;					(* rising edge execute *)
    i_tTimeOut				: TIME := t#10s;  		(* Maximum wait time for reply *)
    i_stControl				: ST_ViciControl;
END_VAR
VAR_OUTPUT
    q_xDone					: BOOL;
    q_xError				: BOOL;
    q_xWarning				: BOOL;					(* set in the event of an unexpected reply *)
    q_xTimeout				: BOOL;
    q_sResult				: STRING(255);
    q_sLastSentString		: ARRAY[1..40] OF STRING;				(* Last String Sent to Serial Device - for debugging *)
    q_sLastReceivedString	: ARRAY[1..40] OF STRING;				(* Last String Received from Serial Device - for debugging *)
    q_stStatus				: ST_ViciStatus;
END_VAR
VAR_IN_OUT
    iq_stSerialRXBuffer 	: ComBuffer;
    iq_stSerialTXBuffer 	: ComBuffer;
END_VAR
VAR
    iReqPosReverse          : INT;
    rtExecute				: R_TRIG;
    iStep					: INT;
    sSendData				: STRING;
    fbViciTransaction		: FB_ViciTransaction;
    (*fbFormatString			: FB_FormatString;*)
    (*fbSplit					: FB_Split255;*)
    asReplyFields			: ARRAY[1..20] OF T_MaxString;
    wChecksum: WORD;
    rtStartIntegration: R_TRIG;
    rtEndReset: R_TRIG;
    sWorking: STRING;
    strResponseExpected: STRING;
END_VAR

(* This function block performs serial transactions with a Vici *)

(* rising edge trigger *)
rtExecute(CLK:= i_xExecute);
IF rtExecute.Q  THEN
    q_xDone	:= FALSE;
    q_xError := FALSE;
    q_xWarning := FALSE;
    q_xTimeout := FALSE;
    q_sResult:= '';
    FBViciTransaction( i_xExecute:= FALSE, iq_stSerialRXBuffer:= iq_stSerialRXBuffer, iq_stSerialTXBuffer:= iq_stSerialTXBuffer );  (* reset *)
    iStep := 10;
END_IF

CASE iStep OF
    0: (* idle *)
        ;

    10: (* Get Position *)
        FBViciTransaction(
            i_xExecute:= TRUE,
            i_iAddress:=i_stControl.iAddress,
            i_sSendData:= 'CP', (*declared postion readback Vici command*)
            i_tTimeOut:= i_tTimeOut,
            iq_stSerialRXBuffer:= iq_stSerialRXBuffer,
            iq_stSerialTXBuffer:= iq_stSerialTXBuffer,
            i_CmdFlag :=FALSE);
        IF FBViciTransaction.q_xError THEN
            q_sResult := CONCAT('in Step 10 serial transaction failed with message: ', FBViciTransaction.q_sResult);
            q_stStatus.xPosValid := FALSE; (* used to signal an invalid readback or control exchange *)
            iStep := 9000;
        ELSIF FBViciTransaction.q_xDone THEN
            q_stStatus.sViciReply := FBViciTransaction.q_sResponseData;
            (* grab the left two characters, they should equal CP *)
            strResponseExpected := CONCAT(INT_TO_STRING( i_stControl.iAddress), 'CP');
            IF LEFT(q_stStatus.sViciReply, 3) <> strResponseExpected (*'1CP'*) THEN
                (*use q-s Result to specify error type*)
                q_sResult := CONCAT(CONCAT('in step 10 unexpected response recieved: ', LEFT(q_stStatus.sViciReply, 3)),CONCAT(' instead of: ', CONCAT(INT_TO_STRING( i_stControl.iAddress), 'CP')));
                    q_xWarning := TRUE;
                (* If they don't equal CP, then error *)
                q_stStatus.xPosValid := FALSE; (* used to signal an invalid readback or control exchange *)
                iStep := 9000;
            (* else then grab the right two characters and convert to INT *)
            ELSE
            sWorking := RIGHT(q_stStatus.sViciReply, 2);
            q_stStatus.iCurrPos := (i_stControl.iPortCount + 1)- STRING_TO_INT(sWorking); (* pass that INT to the q_stStatus.iCurrPos, mirroring positions *)
            q_stStatus.xPosValid := TRUE;
            FBViciTransaction( i_xExecute:= FALSE, iq_stSerialRXBuffer:= iq_stSerialRXBuffer, iq_stSerialTXBuffer:= iq_stSerialTXBuffer, i_CmdFlag :=FALSE);  (* reset *)
            iStep := 5000;
            END_IF
        END_IF


    5000: (* Set position*)
        (* Limit the requested position to the valid possible positions *)
        IF i_stControl.iReqPos > i_stControl.iPortCount OR i_stControl.iReqPos < 1 THEN
            q_sResult := CONCAT('in step 5000 port range exceeded: ',FBViciTransaction.q_sResponseData);
            i_stControl.iReqPos := LIMIT(1, i_stControl.iReqPos, i_stControl.iPortCount);
        END_IF
        (* Mirror the "clock" value across the vertical axis of symmetry *)
        iReqPosReverse := (i_stControl.iPortCount + 1) - i_stControl.iReqPos;
        IF q_stStatus.iReqPos <> i_stControl.iReqPos THEN

            // Move actuator to new position via the shortest path
            sSendData := CONCAT('GO', INT_TO_STRING(iReqPosReverse));

            FBViciTransaction(
                i_xExecute:= TRUE,
                i_sSendData:= sSendData,
                i_tTimeOut:= i_tTimeOut,
                i_iAddress:=i_stControl.iAddress,
                iq_stSerialRXBuffer:= iq_stSerialRXBuffer,
                iq_stSerialTXBuffer:= iq_stSerialTXBuffer,
                i_CmdFlag:=TRUE);
            IF FBViciTransaction.q_xError THEN
                q_sResult := CONCAT('in Step 5000 serial transaction failed with message: ', FBViciTransaction.q_sResult);
                iStep := 9000;
            ELSIF FBViciTransaction.q_xDone THEN
                FBViciTransaction(
                     i_xExecute:= FALSE,
                    iq_stSerialRXBuffer:= iq_stSerialRXBuffer,
                    iq_stSerialTXBuffer:= iq_stSerialTXBuffer,
                    i_CmdFlag:=FALSE );  (* reset *)
                q_stStatus.iReqPos := i_stControl.iReqPos;
                iStep := 8000;
            END_IF
        ELSE
            iStep := 8000;
        END_IF


    8000: (* done *)
        q_xDone := TRUE;
        IF q_sResult = '' THEN
            q_sResult := 'Success';
        END_IF
        IF  i_xExecute = FALSE THEN
            q_xDone:= FALSE;
            iStep := 0;
        END_IF

    9000:
        _A_ClearStatus();
        q_xTimeout := FBViciTransaction.q_xTimeout;
        q_xError := TRUE;


END_CASE

q_sLastSentString := FBViciTransaction.q_sLastSentString;
q_sLastReceivedString := FBViciTransaction.q_sLastReceivedString;

ACTION _A_ClearStatus:
q_stStatus.sViciReply := '';
END_ACTION

END_FUNCTION_BLOCK
